FUNCTION_BLOCK HVglobalError (* Basic Function Block Type *)
  (* Standard: 61499-2 *)
  (* Version 0.0, 11/17/2015, bglatz, nxtControl GmbH, Template *)
  PACKAGE Loytec.HVAC;
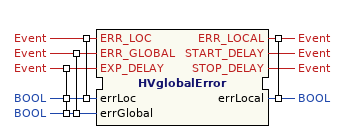
  EVENT_INPUT
    ERR_LOC WITH errLoc; (* Normal Execution Request *)
    ERR_GLOBAL WITH errGlobal;
    EXP_DELAY WITH errLoc, errGlobal;
  END_EVENT
  EVENT_OUTPUT
    ERR_LOCAL WITH errLocal; (* Execution Confirmation *)
    START_DELAY;
    STOP_DELAY;
  END_EVENT
  VAR_INPUT
    errLoc : BOOL;
    errGlobal : BOOL;
  END_VAR
  VAR_OUTPUT
    errLocal : BOOL := FALSE; (* Output event qualifier *)
  END_VAR
  VAR
    timerRun : BOOL := FALSE;
  END_VAR
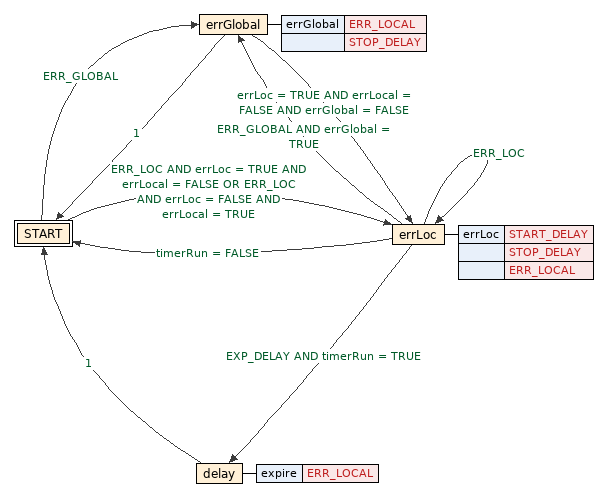
  EC_STATES
    START; (* Initial State *)
    errLoc : errLoc -> START_DELAY, -> STOP_DELAY, -> ERR_LOCAL;
    delay : expire -> ERR_LOCAL;
    errGlobal : errGlobal -> ERR_LOCAL, -> STOP_DELAY;
  END_STATES
  EC_TRANSITIONS
    START TO errLoc := ERR_LOC AND errLoc = TRUE AND errLocal = FALSE OR ERR_LOC AND errLoc = FALSE AND errLocal = TRUE;
    errLoc TO delay := EXP_DELAY AND timerRun = TRUE;
    errLoc TO START := timerRun = FALSE;
    errLoc TO errLoc := ERR_LOC;
    delay TO START := 1;
    START TO errGlobal := ERR_GLOBAL;
    errLoc TO errGlobal := ERR_GLOBAL AND errGlobal = TRUE;
    errGlobal TO errLoc := errLoc = TRUE AND errLocal = FALSE AND errGlobal = FALSE;
    errGlobal TO START := 1;
  END_TRANSITIONS
  ALGORITHM errLoc IN ST:
VAR
	tmp : BOOL;
END_VAR;

tmp := errLocal;

ERR_LOC := FALSE;

errLocal := FALSE;

IF errLoc = TRUE THEN
	IF timerRun = FALSE THEN
		timerRun := TRUE;
		STOP_DELAY := FALSE;
	ELSE
		STOP_DELAY := FALSE;
		START_DELAY := FALSE;
	END_IF;
ELSE
	IF timerRun = TRUE THEN
		timerRun := FALSE;
		START_DELAY := FALSE;
	ELSE
		START_DELAY := FALSE;
		STOP_DELAY := FALSE;
	END_IF;
END_IF;

IF tmp = errLocal THEN
	ERR_LOCAL := FALSE;
END_IF;
  END_ALGORITHM
  ALGORITHM expire IN ST:
timerRun := FALSE;

errLocal := TRUE;
  END_ALGORITHM
  ALGORITHM errGlobal IN ST:
VAR
	tmp : BOOL;
END_VAR;

tmp := errLocal;

ERR_GLOBAL := FALSE;

(* from armed timer *)
IF timerRun = TRUE THEN
	timerRun := FALSE;
	errLocal := FALSE;
ELSE
	(* from idle state *)
	IF errGlobal = TRUE THEN
		errLocal := FALSE;
	END_IF;
	STOP_DELAY := FALSE;
END_IF;

IF tmp = errLocal THEN
	ERR_LOCAL := FALSE;
END_IF;
  END_ALGORITHM
END_FUNCTION_BLOCK
